FUNCTION WORD_TO_BYTES
  (* Standard: 61499-1 *)
  (* Version 1.0, 2024-02-22, franz *)
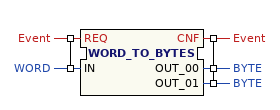
  EVENT_INPUT
    REQ WITH IN; (* Normal Execution Request *)
  END_EVENT
  EVENT_OUTPUT
    CNF WITH OUT_00, OUT_01; (* Execution Confirmation *)
  END_EVENT
  VAR_INPUT
    IN : WORD; (* WORD Input *)
  END_VAR
  VAR_OUTPUT
    OUT_00 : BYTE; (* BYTE 00 *)
    OUT_01 : BYTE; (* BYTE 01 *)
  END_VAR
  BODY IN ST:
FUNCTION WORD_TO_BYTES

VAR_INPUT
	IN : WORD;    // WORD Input
END_VAR

VAR_OUTPUT
	OUT_00 : BYTE;    // BYTE 00
	OUT_01 : BYTE;    // BYTE 01
END_VAR

(* this Function extracts the 2 BYTE from a word *)
OUT_00 := WORD_TO_BYTE(IN AND WORD_BYTE_00);
OUT_01 := WORD_TO_BYTE(SHR(IN AND WORD_BYTE_01, 8));

END_FUNCTION
  END_BODY
END_FUNCTION
